// Mitsubishi GX Works2 project: Test bisa dicoba coba   PLC: FX1N/FX1NC
// FX3S_Terco_Awal

PROGRAM MAIN  // ladder awal
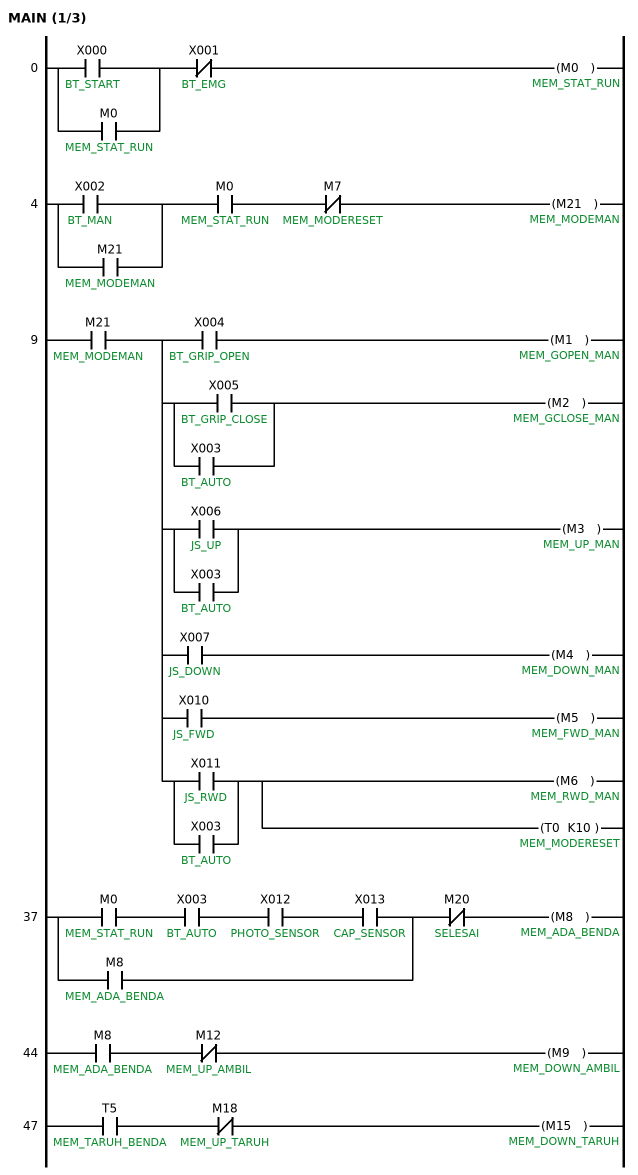
0     LD      X000  ; BT_START
      OR      M0  ; MEM_STAT_RUN
      ANI     X001  ; BT_EMG
      OUT     M0  ; MEM_STAT_RUN
4     LD      X002  ; BT_MAN
      OR      M21  ; MEM_MODEMAN
      AND     M0  ; MEM_STAT_RUN
      ANI     M7  ; MEM_MODERESET
      OUT     M21  ; MEM_MODEMAN
9     LD      M21  ; MEM_MODEMAN
      MPS
      AND     X004  ; BT_GRIP_OPEN
      OUT     M1  ; MEM_GOPEN_MAN
      MRD
      LD      X005  ; BT_GRIP_CLOSE
      OR      X003  ; BT_AUTO
      ANB
      OUT     M2  ; MEM_GCLOSE_MAN
      MRD
      LD      X006  ; JS_UP
      OR      X003  ; BT_AUTO
      ANB
      OUT     M3  ; MEM_UP_MAN
      MRD
      AND     X007  ; JS_DOWN
      OUT     M4  ; MEM_DOWN_MAN
      MRD
      AND     X010  ; JS_FWD
      OUT     M5  ; MEM_FWD_MAN
      MPP
      LD      X011  ; JS_RWD
      OR      X003  ; BT_AUTO
      ANB
      OUT     M6  ; MEM_RWD_MAN
      OUT     T0 K10  ; MEM_MODERESET
37    LD      M0  ; MEM_STAT_RUN
      AND     X003  ; BT_AUTO
      AND     X012  ; PHOTO_SENSOR
      AND     X013  ; CAP_SENSOR
      OR      M8  ; MEM_ADA_BENDA
      ANI     M20  ; SELESAI
      OUT     M8  ; MEM_ADA_BENDA
44    LD      M8  ; MEM_ADA_BENDA
      ANI     M12  ; MEM_UP_AMBIL
      OUT     M9  ; MEM_DOWN_AMBIL
47    LD      T5  ; MEM_TARUH_BENDA
      ANI     M18  ; MEM_UP_TARUH
      OUT     M15  ; MEM_DOWN_TARUH
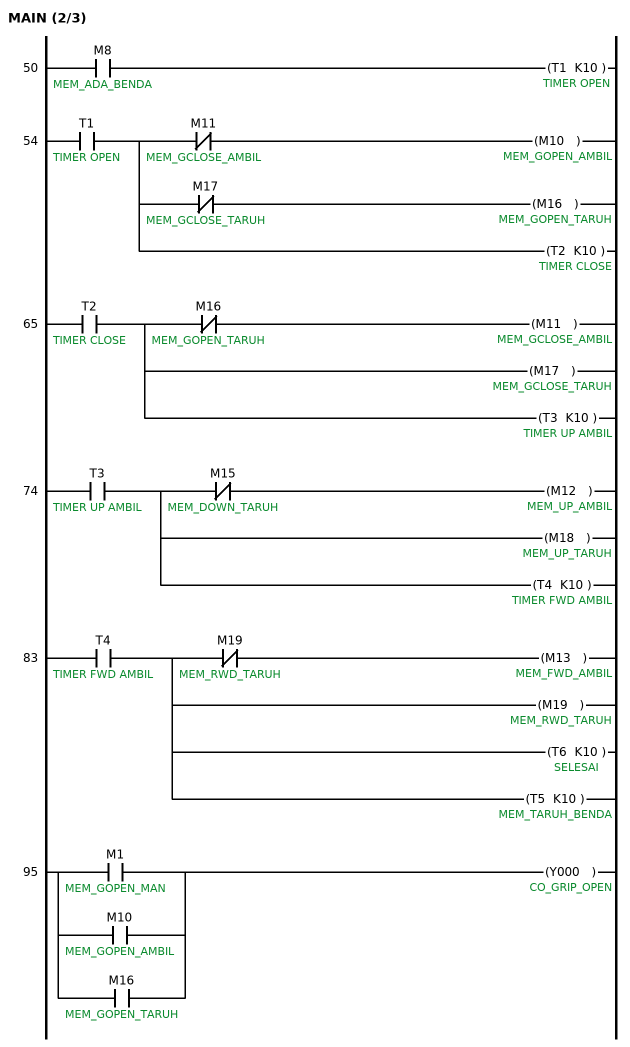
50    LD      M8  ; MEM_ADA_BENDA
      OUT     T1 K10  ; TIMER OPEN
54    LD      T1  ; TIMER OPEN
      MPS
      ANI     M11  ; MEM_GCLOSE_AMBIL
      OUT     M10  ; MEM_GOPEN_AMBIL
      MRD
      ANI     M17  ; MEM_GCLOSE_TARUH
      OUT     M16  ; MEM_GOPEN_TARUH
      MPP
      OUT     T2 K10  ; TIMER CLOSE
65    LD      T2  ; TIMER CLOSE
      MPS
      ANI     M16  ; MEM_GOPEN_TARUH
      OUT     M11  ; MEM_GCLOSE_AMBIL
      MPP
      OUT     M17  ; MEM_GCLOSE_TARUH
      OUT     T3 K10  ; TIMER UP AMBIL
74    LD      T3  ; TIMER UP AMBIL
      MPS
      ANI     M15  ; MEM_DOWN_TARUH
      OUT     M12  ; MEM_UP_AMBIL
      MPP
      OUT     M18  ; MEM_UP_TARUH
      OUT     T4 K10  ; TIMER FWD AMBIL
83    LD      T4  ; TIMER FWD AMBIL
      MPS
      ANI     M19  ; MEM_RWD_TARUH
      OUT     M13  ; MEM_FWD_AMBIL
      MPP
      OUT     M19  ; MEM_RWD_TARUH
      OUT     T6 K10  ; SELESAI
      OUT     T5 K10  ; MEM_TARUH_BENDA
95    LD      M1  ; MEM_GOPEN_MAN
      OR      M10  ; MEM_GOPEN_AMBIL
      OR      M16  ; MEM_GOPEN_TARUH
      OUT     Y000  ; CO_GRIP_OPEN
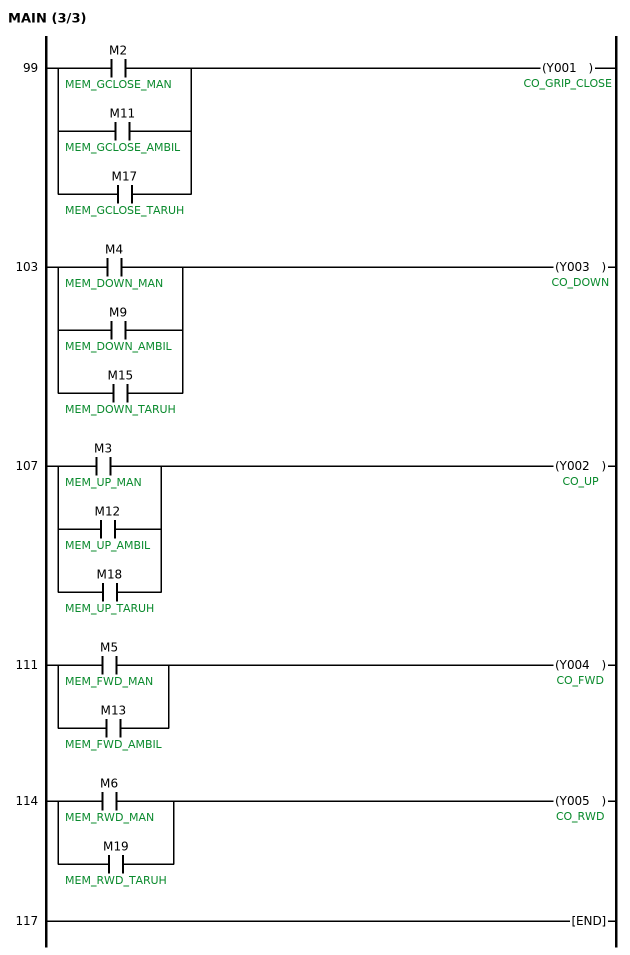
99    LD      M2  ; MEM_GCLOSE_MAN
      OR      M11  ; MEM_GCLOSE_AMBIL
      OR      M17  ; MEM_GCLOSE_TARUH
      OUT     Y001  ; CO_GRIP_CLOSE
103   LD      M4  ; MEM_DOWN_MAN
      OR      M9  ; MEM_DOWN_AMBIL
      OR      M15  ; MEM_DOWN_TARUH
      OUT     Y003  ; CO_DOWN
107   LD      M3  ; MEM_UP_MAN
      OR      M12  ; MEM_UP_AMBIL
      OR      M18  ; MEM_UP_TARUH
      OUT     Y002  ; CO_UP
111   LD      M5  ; MEM_FWD_MAN
      OR      M13  ; MEM_FWD_AMBIL
      OUT     Y004  ; CO_FWD
114   LD      M6  ; MEM_RWD_MAN
      OR      M19  ; MEM_RWD_TARUH
      OUT     Y005  ; CO_RWD
117   END
END_PROGRAM
